{attribute 'no_explicit_call' := 'Contactor is a CLASS and must be accessed using methods or properties'}
FUNCTION_BLOCK Contactor
VAR
	output				AT %Q*: BOOL;
END_VAR

METHOD SwitchOff
VAR_INPUT
END_VAR
output   := false;
END_METHOD

METHOD SwitchOn
VAR_INPUT
END_VAR
output   := true;
END_METHOD

END_FUNCTION_BLOCK

(* stored: Version 1.1.0.1, ProductVersion 3.1.4024.11
   POU Contactor: Id {664e749d-a50b-4bbd-bd24-e8f436436cd9}, SpecialFunc None
   Method SwitchOff: Id {ae9d30a0-94a1-419a-ad1c-2911e0c12fb3}
   Method SwitchOn: Id {18d83911-4b9c-43e2-8c44-46ace6308946} *)
